// TIA Portal V21 export
DATA_BLOCK "DB627"   // DB627
TITLE = SCREEN PROCESS VALUE
{ S7_Optimized_Access := 'FALSE' }
// stored: AutoNumber false
   VAR
      RinseTimeSv : Int;
      RinseTimePv : DInt;
      FillTimeSv : DInt;
      FillTimePv : DInt;
      RepSv : Int;
      RepPv : Int;
      FillQtySv : Real;
      FillQtyPv : Real;
      MixingSv : Int;
      MixingPv : DInt;
      SdSv : Int;
      SdPv : DInt;
      APSv : Int;
      ApPv : DInt;
      ApReleaseTimeSv : Int;
      ApReleaseTimePv : DInt;
      CurrentStepNo : Int;
      CycleStatus : String[60];
      StepStatus : String[60];
      ApSetPressureSv : Real;
      ApSetPressurePv : Real;
      CombineAPSv : Int;
      CombineApPv : DInt;
      CombineApReleaseTimeSv : Int;
      CombineApReleaseTimePv : DInt;
      DosingTimePv : DInt;
      PulsingTimeSv : Int;
      RecirculationSv : Int;
      RecirculationPv : DInt;
      ConductivitySv : Real;
      ConductivityPv : Real;
   END_VAR
BEGIN
END_DATA_BLOCK
